// TIA Portal V19 export
TYPE "MES_Msg_Receive_Topic2xx_Err"
// stored: Access Published
   STRUCT
      Recive_MSG200 { ExternalAccessible := 'False'; ExternalVisible := 'False'; ExternalWritable := 'False'} : "MES_Err_&_Msg";
      Recive_MSG210 { ExternalAccessible := 'False'; ExternalVisible := 'False'; ExternalWritable := 'False'} : "MES_Err_&_Msg";
      Recive_MSG212 { ExternalAccessible := 'False'; ExternalVisible := 'False'; ExternalWritable := 'False'} : "MES_Err_&_Msg";
      Send_MSG201_Follow_MSG200 { ExternalAccessible := 'False'; ExternalVisible := 'False'; ExternalWritable := 'False'} : "MES_Err_&_Msg";
      Send_MSG211_Follow_MSG210 { ExternalAccessible := 'False'; ExternalVisible := 'False'; ExternalWritable := 'False'} : "MES_Err_&_Msg";
   END_STRUCT;
END_TYPE
